INTERFACE I_Observable EXTENDS I_Observer

{attribute 'OPC.UA.DA.Property' := '1'}
{attribute 'monitoring' := 'call'}
PROPERTY P_Length : DINT
GET
END_GET
END_PROPERTY

METHOD M_Detach : BOOL
VAR_INPUT
	Object: 	I_Component;
END_VAR
END_METHOD

METHOD M_Attach : BOOL
VAR_INPUT
	Object: 	I_Component;
END_VAR
END_METHOD

END_INTERFACE

(* stored: Version 1.1.0.1
   Itf I_Observable: Id {af54216d-3f5e-4287-8176-18b478632bd5}
   Property P_Length: Id {b558abeb-888e-0699-2ea6-95610585a3fc}
   Get Get: Id {343bf9e3-5746-0336-07c3-d87ab710257c}
   Method M_Detach: Id {e09cef4f-639e-464f-affe-bde457fdaa63}
   Method M_Attach: Id {e1012f71-0b48-4ada-ba34-823492d9c2fe} *)
